// TIA Portal V19 export
FUNCTION "Move MAC" : Void   // FC11, LAD
{ S7_Optimized_Access := 'TRUE' }
// stored: SetENOAutomatically false
   VAR_INPUT
      InMAC : Array[0..5] of Byte;
   END_VAR
   VAR_OUTPUT
      OutMAC : Array[0..5] of Byte;
   END_VAR
BEGIN

REGION Network 1
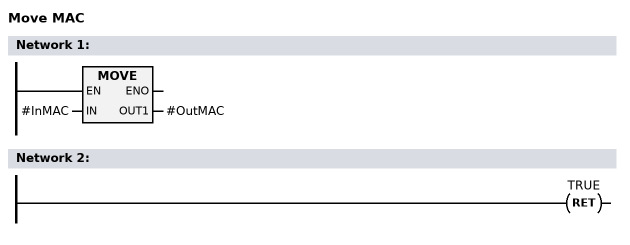
   RUNG wire#powerrail
      Move(in := #InMAC, out1 => #OutMAC)
   END_RUNG
   // the same network as SCL:
   #OutMAC := #InMAC;
END_REGION

REGION Network 2
   RUNG wire#powerrail
      ReturnCoil( TRUE )
   END_RUNG
   // the same network as SCL:
   ENO := TRUE;
   RETURN;
END_REGION
END_FUNCTION
